GLOBALCONSTANTS motorNummer (* Motor-Identitaet als SINT (0 = keiner, 1..6 = Mx), fuer AnlagenSequenz_06.TRANSIT_MOTOR, s. KONZEPT_Anlagensequenz.md *)
  (* Standard: 61499-1; Description: Copyright (c) 2026 HR Agrartechnik GmbH This program and the accompanying materials are made available under the terms of the Eclipse Public License 2.0 which is available at https://www.eclipse.org/legal/epl-2.0/ SPDX-License-Identifier: EPL-2.0 *)
  (* Version 1.0, 2026-08-25, Franz Höpfinger, HR Agrartechnik GmbH *)
  PACKAGE logiBUS::utils::sequence::const;
  VAR_GLOBAL CONSTANT
    MOTOR_KEINER : SINT := SINT#0; (* kein Motor *)
    MOTOR_M1 : SINT := SINT#1; (* Motor 1 *)
    MOTOR_M2 : SINT := SINT#2; (* Motor 2 *)
    MOTOR_M3 : SINT := SINT#3; (* Motor 3 *)
    MOTOR_M4 : SINT := SINT#4; (* Motor 4 *)
    MOTOR_M5 : SINT := SINT#5; (* Motor 5 *)
    MOTOR_M6 : SINT := SINT#6; (* Motor 6 *)
  END_VAR
END_GLOBALCONSTANTS
